{attribute 'qualified_only'}
{attribute 'strict'}
TYPE E_PopupSymbol :
(
	ePopupSymbolNone := 0,
	ePopupSymbolOk,
	ePopupSymbolNok
);
END_TYPE

(* stored: Version 1.1.0.1, ProductVersion 3.1.4024.11
   DUT E_PopupSymbol: Id {30f7cfb1-a634-41b9-80a8-e8c33579d4f4} *)
